INTERFACE I_Job EXTENDS I_Debug

METHOD Run : TaskState
END_METHOD

END_INTERFACE

(* stored: Version 1.1.0.1
   Itf I_Job: Id {87a9768c-0425-48bc-8261-07f4f0c86d1c}
   Method Run: Id {c44a7cd6-6690-4a0e-afed-d33e68feddb0} *)
